// TIA Portal V21 export
TYPE "switchgearStatus"
   STRUCT
      ready : Bool;
      run : Bool;
      operation : Bool;
      alm : Bool;
      unackAlm : Bool;
   END_STRUCT;
END_TYPE
